// TIA Portal V18 export
// export: Created 2025-12-01T17:53:07.3121448Z, ExportSetting None, DisplayName Totally Integrated Automation Portal, DisplayVersion V18 Update 5, DisplayName TIA Portal Openness, DisplayVersion V18 Update 5, DisplayName TIA Portal Teamcenter Gateway, DisplayVersion V18, DisplayName TIA Portal Version Control Interface, DisplayVersion V18, DisplayName STEP 7 Professional, DisplayVersion V18 Update 5, DisplayName STEP 7 Safety, DisplayVersion V18, DisplayName WinCC Professional, DisplayVersion V18 Update 5
Screen "300Main"  1280x800, Number=300, Template=T1
  ScreenLayer "Layer_0"
    Button "按钮_6" at 384,725 size 128x75  PictureOff=向左箭头_0, StyleItem=BtnFunction20, TextOff="报警确认 / Alarm confirm / Poplach potvrdiť"
      on Click: AlarmViewAcknowledgeAlarm(Screen object := 报警视图_1)
    Button "按钮_7" at 256,725 size 128x75  PictureOff=向左箭头_0, StyleItem=BtnNormal20, TextOff="历史报警 / Alarm history / Alarm Geschichte"
      on Click: ActivateScreen(Screen name := 310History, Object number := 0); SetTag(Tag := Sys_VersionManagement_HMIPageID, Value := 310)
    Button "按钮_1" at 128,725 size 128x75  PictureOff=向左箭头_0, StyleItem=BtnActive20, TextOff="当前报警 / Alarm / Poplach"
      on Click: ActivateScreen(Screen name := , Object number := 0); SetTag(Tag := Sys_VersionManagement_HMIPageID, Value := 300)
